FUNCTION_BLOCK CSWI_Logic (* Basic Function Block Type *)
  (* Standard: 61499-2 *)
  (* Version 0.0, 12/11/2023, Cheyan, Schneider Electric, Template *)
  PACKAGE Main;
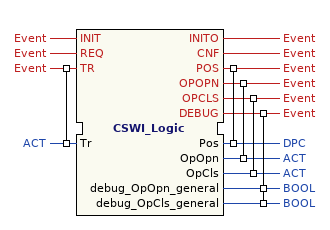
  EVENT_INPUT
    INIT; (* Initialization Request *)
    REQ; (* Normal Execution Request *)
    TR WITH Tr;
  END_EVENT
  EVENT_OUTPUT
    INITO; (* Initialization Confirm *)
    CNF; (* Execution Confirmation *)
    POS WITH Pos;
    OPOPN WITH OpOpn;
    OPCLS WITH OpCls;
    DEBUG WITH debug_OpOpn_general, debug_OpCls_general;
  END_EVENT
  VAR_INPUT
    Tr : ACT; (* Input event qualifier *)
  END_VAR
  VAR_OUTPUT
    Pos : DPC;
    OpOpn : ACT;
    OpCls : ACT;
    debug_OpOpn_general : BOOL;
    debug_OpCls_general : BOOL;
  END_VAR
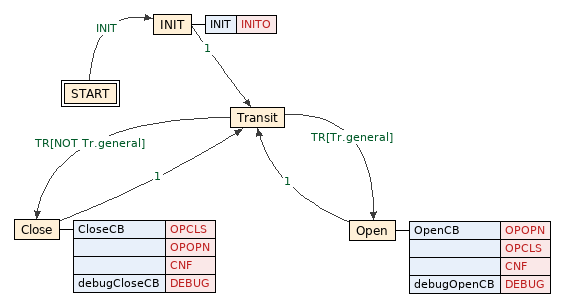
  EC_STATES
    START; (* Initial State *)
    INIT : INIT -> INITO; (* Initialization *)
    Open : OpenCB -> OPOPN, -> OPCLS, -> CNF, debugOpenCB -> DEBUG; (* Normal execution *)
    Transit;
    Close : CloseCB -> OPCLS, -> OPOPN, -> CNF, debugCloseCB -> DEBUG;
  END_STATES
  EC_TRANSITIONS
    START TO INIT := INIT;
    INIT TO Transit := 1;
    Transit TO Open := TR[Tr.general];
    Open TO Transit := 1;
    Transit TO Close := TR[NOT Tr.general];
    Close TO Transit := 1;
  END_TRANSITIONS
  ALGORITHM INIT IN ST: (* Initialization algorithm Initializing the start state of the CB to the "Closed" State *)
;

OpOpn.general := FALSE;
OpCls.general := TRUE;
  END_ALGORITHM
  ALGORITHM OpenCB IN ST: (* Normally executed algorithm To close the circuit breaker, set OpOpn_general to true and OpCls_general to false *)
;

Pos.stVal := Main.stVal#item2;
OpOpn.general := TRUE;
OpCls.general := FALSE;
  END_ALGORITHM
  ALGORITHM CloseCB IN ST: (* To open the circuit breaker, set OpOpn_general to false and OpCls_general to true *)
;

Pos.stVal := Main.stVal#item3;
OpOpn.general := FALSE;
OpCls.general := TRUE;
  END_ALGORITHM
  ALGORITHM debugOpenCB IN ST:
;

debug_OpOpn_general := TRUE;
debug_OpCls_general := FALSE;
  END_ALGORITHM
  ALGORITHM debugCloseCB IN ST:
;

debug_OpOpn_general := FALSE;
debug_OpCls_general := TRUE;
  END_ALGORITHM
END_FUNCTION_BLOCK
